{attribute 'GeneratedUsingTerminal: AX8108-0100-0101-0101'}
{attribute addProperty BoxType "AX8108-0100-0101-0101"}
{attribute addProperty Id "FSOEAT %Q*FSOE_6A82EB9321"}
{attribute addProperty CRC "1896473840"}
{attribute addProperty Size "21"}
TYPE FSoE_Slave_Connection_1_Master_Message_7109E4F0 EXTENDS OutputBase_10CEE7DE :
STRUCT
	{attribute addProperty Name "FSOE"}
	FSOE AT %Q* : FSOE_6A82EB93;
END_STRUCT
END_TYPE

(* stored: Version 1.2.0.0, ProductVersion 3.1.4024.9
   DUT FSoE_Slave_Connection_1_Master_Message_7109E4F0: Id {008f0315-f2b1-471a-a734-24fb97dc9ccf} *)
